INTERFACE I_Name

PROPERTY Name : STRING
GET
END_GET
SET
END_SET
END_PROPERTY

END_INTERFACE

(* stored: Version 1.1.0.1, ProductVersion 3.1.4024.12
   Itf I_Name: Id {74b67812-4e6d-4c4f-87a7-f91d056aa0f4}
   Property Name: Id {405bec32-6394-4c95-a111-2649d28c22d5}
   Get Get: Id {121a5791-58ec-40aa-be85-dbc1878e5d76}
   Set Set: Id {83a33692-929f-4161-a571-af2d8975242a} *)
